(* works for 901 with Ethercat interface*)
{attribute 'no_check'}
FUNCTION_BLOCK FB_901_ECAT  EXTENDS FB_GaugeBase
VAR_INPUT
END_VAR
VAR_OUTPUT
	{attribute 'pytmc' := '
    pv: 
	'}
	PG	: ST_VG;
END_VAR
VAR_IN_OUT
	
END_VAR
VAR
	bInit: BOOL:= TRUE;(*IO*)
	xPress_OK AT%I* : BOOL;
	xOverrange AT%I* : BOOL;
	xUnderrange AT%I* : BOOL; 
	i_iPRESS_R AT%I* : REAL; // input Pressure // Link to analog Input
	bWcstate AT%I* : BOOL; // 0: date valid, 1: date invalid
	
END_VAR

(* Standard MKS 9XX series conversion *)
(* works for 901 with Ethercat interface*)
// no div by zero
PG.rPRESS :=i_iPRESS_R;
PG.xPRESS_OK := xPress_OK and NOT bWcstate ;
IF xPress_OK and NOT bWcstate THEN
	PG.xPRESS_OK := TRUE;
	PG.eState := Valid; //Press OK
ELSIF xOverrange and NOT bWcstate THEN
	PG.xPRESS_OK := FALSE;
	PG.eState := OoR;
ELSIF xUnderrange and NOT bWcstate THEN
	PG.xPRESS_OK := FALSE;
	PG.eState := PressInvalid;

END_IF



(*Logger*)
ACT_Logger();
(* Soft IO Mapping*)
ACT_IO();

ACTION ACT_Init:
IF (bInit) THEN
	bInit := False;
	
	//set pressure units to Torr
	// value 0x00A10000 SDO index 0xf840, si 0x01 UDINT
END_IF
END_ACTION

ACTION ACT_IO:

IF PG.xPRESS_OK THEN
  	PG.i_iPRESS_R := REAL_TO_INT(i_iPRESS_R);
ELSE
	PG.rPRESS := 0.0;
END_IF
PG.sPath := sPath;
END_ACTION

ACTION ACT_Logger:

//STATE Logger  
IF ePrevState <> PG.eState THEN
	  CASE PG.eState OF
		ValidHi:
			fbLogger(sMsg:='Gauge pressure valid high.', eSevr:=TcEventSeverity.Info);
		ValidLo:
			fbLogger(sMsg:='Gauge pressure valid low.', eSevr:=TcEventSeverity.Info);
		Valid:
			fbLogger(sMsg:='Gauge pressure valid.', eSevr:=TcEventSeverity.Info);
  		GaugeDisconnected:
			fbLogger(sMsg:='Gauge Disconnected.', eSevr:=TcEventSeverity.Critical);
		PressInvalid:
			fbLogger(sMsg:='Gauge pressure invalid.', eSevr:=TcEventSeverity.Warning);
		OoR:
			fbLogger(sMsg:='Gauge pressure out of range.', eSevr:=TcEventSeverity.Warning);
		Starting:
			fbLogger(sMsg:='Gauge starting.', eSevr:=TcEventSeverity.Info);
	  END_CASE
	  ePrevState := PG.eState;  
  END_IF
END_ACTION

END_FUNCTION_BLOCK

(* stored: Version 1.1.0.1, ProductVersion 3.1.4022.18
   POU FB_901_ECAT: Id {84706132-589d-4d51-8b00-ab55510b97b2}, SpecialFunc None
   Action ACT_Init: Id {79fc3e26-9526-4887-bb81-9ff0cb209da7}
   Action ACT_IO: Id {afe7d8e6-827d-4f4d-895b-401bfcc2f6f0}
   Action ACT_Logger: Id {4887216a-c77e-43cb-a418-2b8dd97c0d8a} *)
